PROGRAM MAIN
VAR
END_VAR

END_PROGRAM

(* stored: Version 1.1.0.1
   POU MAIN: Id {b8490017-7447-42a1-9034-331e661ac42b} *)
